PROGRAM P_MotionControl
VAR
	

//////Dette brukes i det nye////////////

//Enable Motion
	bAutoEnable_PC 							: BOOL;
	bManualEnable_PC 						: BOOL; 
	bAutoEnable_SC 							: BOOL; 
	bManualEnable_SC					    : BOOL;
	bCombinationEnable						: BOOL;

/////////// Function blocks////////// 
	
	//Enable Motion
	fbEnableMotion							: FB_Enable_Motion;
	
	//Primary Control
	fbManual_PC								: FB_Manual_PC;
	fbAuto_PC								: FB_Auto_PC;
	
	//Secondary Control
	fbManual_SC								: FB_Manual_SC;
	fbAuto_SC								: FB_Auto_SC;

	//Combination
	fbCombination							: FB_Auto_Combination;

	//Endstop
	fbEndstop								: FB_EndStop;

	//MUX
	fbMUX_selector							: FB_MUX_selector;

/////OutPut Variables////
	fPCV_MPC							: LREAL;
	fSCV_MPC							: LREAL;
	
	fPCV_APC							: LREAL;
	fSCV_APC							: LREAL;
	
	fPCV_MSC							: LREAL;
	fSCV_MSC							: LREAL;
	
	fPCV_ASC							: LREAL;
	fSCV_ASC							: LREAL;
	
	fPCV_combi							: LREAL;
	fSCV_combi							: LREAL;
	
	//After MUX
	fPCV							: LREAL;
	fSCV							: LREAL;
	fPCV_norm_input					: LREAL;
	fSCV_norm_input					: LREAL;
	
	
//ValveOutputs
fbOutputs							: FB_Outputs;
fPCV_raw							: INT;
fSCV_raw							: INT;
	
END_VAR

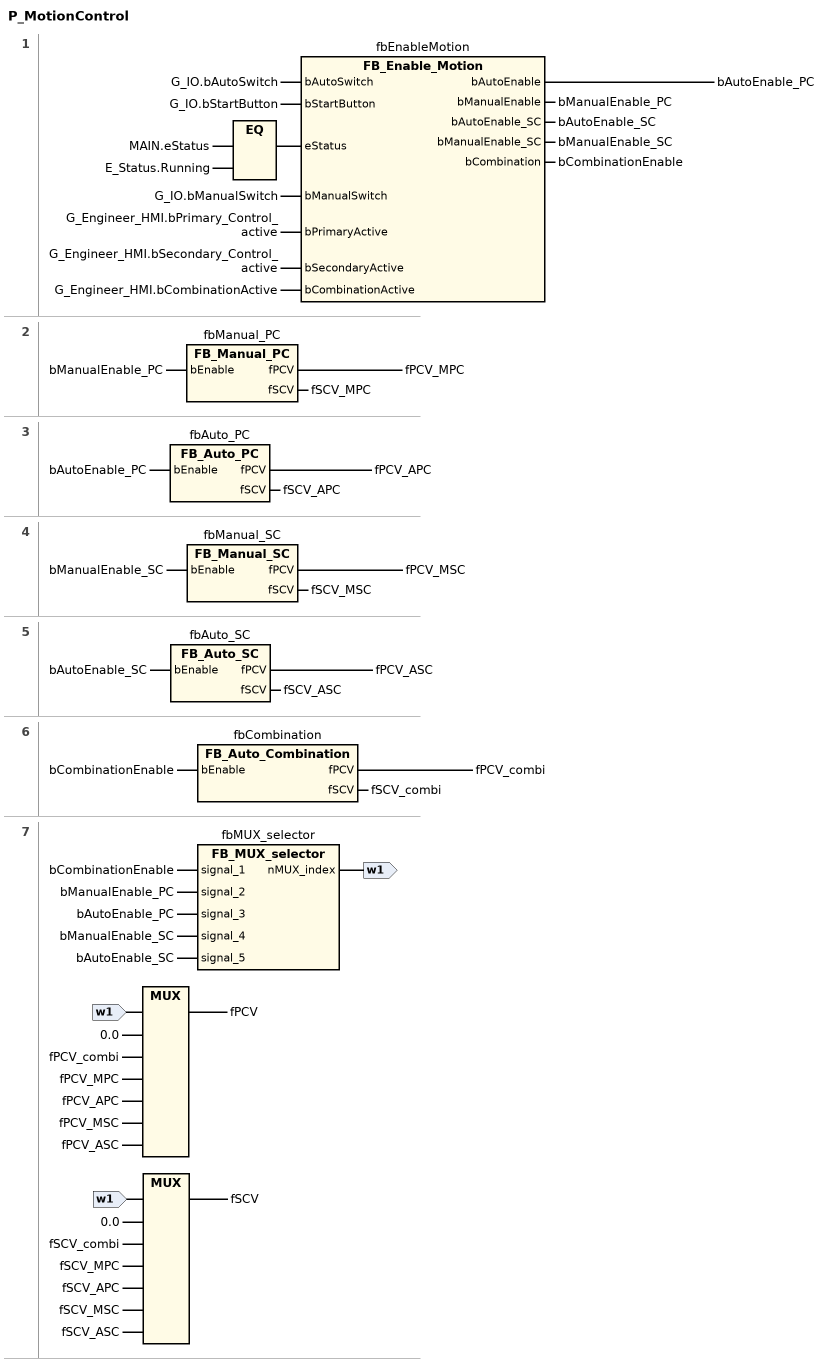
// NETWORK 1
fbEnableMotion(
    bAutoSwitch := G_IO.bAutoSwitch,
    bStartButton := G_IO.bStartButton,
    eStatus := MAIN.eStatus = E_Status.Running,
    bManualSwitch := G_IO.bManualSwitch,
    bPrimaryActive := G_Engineer_HMI.bPrimary_Control_active,
    bSecondaryActive := G_Engineer_HMI.bSecondary_Control_active,
    bCombinationActive := G_Engineer_HMI.bCombinationActive,
    bManualEnable => bManualEnable_PC,
    bAutoEnable_SC => bAutoEnable_SC,
    bManualEnable_SC => bManualEnable_SC,
    bCombination => bCombinationEnable); // FB_Enable_Motion
bAutoEnable_PC := fbEnableMotion.bAutoEnable;

// NETWORK 2
fbManual_PC(bEnable := bManualEnable_PC, fSCV => fSCV_MPC); // FB_Manual_PC
fPCV_MPC := fbManual_PC.fPCV;

// NETWORK 3
fbAuto_PC(bEnable := bAutoEnable_PC, fSCV => fSCV_APC); // FB_Auto_PC
fPCV_APC := fbAuto_PC.fPCV;

// NETWORK 4
fbManual_SC(bEnable := bManualEnable_SC, fSCV => fSCV_MSC); // FB_Manual_SC
fPCV_MSC := fbManual_SC.fPCV;

// NETWORK 5
fbAuto_SC(bEnable := bAutoEnable_SC, fSCV => fSCV_ASC); // FB_Auto_SC
fPCV_ASC := fbAuto_SC.fPCV;

// NETWORK 6
fbCombination(bEnable := bCombinationEnable, fSCV => fSCV_combi); // FB_Auto_Combination
fPCV_combi := fbCombination.fPCV;

// NETWORK 7
fbMUX_selector(
    signal_1 := bCombinationEnable,
    signal_2 := bManualEnable_PC,
    signal_3 := bAutoEnable_PC,
    signal_4 := bManualEnable_SC,
    signal_5 := bAutoEnable_SC); // FB_MUX_selector
fPCV := MUX(fbMUX_selector.nMUX_index, 0.0, fPCV_combi, fPCV_MPC, fPCV_APC, fPCV_MSC, fPCV_ASC);
fSCV := MUX(fbMUX_selector.nMUX_index, 0.0, fSCV_combi, fSCV_MPC, fSCV_APC, fSCV_MSC, fSCV_ASC);

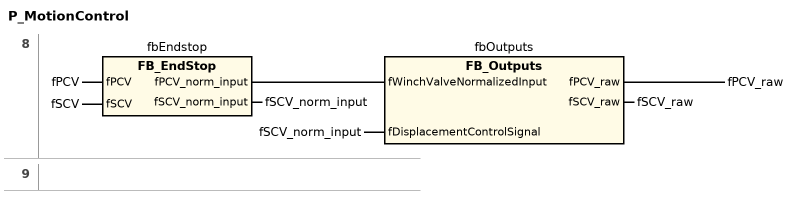
// NETWORK 8
fbEndstop(fPCV := fPCV, fSCV := fSCV, fSCV_norm_input => fSCV_norm_input); // FB_EndStop
fbOutputs(
    fWinchValveNormalizedInput := fbEndstop.fPCV_norm_input,
    fDisplacementControlSignal := fSCV_norm_input,
    fSCV_raw => fSCV_raw); // FB_Outputs
fPCV_raw := fbOutputs.fPCV_raw;

// NETWORK 9

END_PROGRAM

(* stored: Version 1.1.0.1
   POU P_MotionControl: Id {379b28a6-997a-4ccf-86a8-6ee28f5b3d59}, SpecialFunc None *)
